// TIA Portal V17 export
// export: Created 2023-02-26T22:59:49.9931463Z, ExportSetting WithDefaults, DisplayName Totally Integrated Automation Portal, DisplayVersion V17, DisplayName TIA Portal Openness, DisplayVersion V17, DisplayName TIA Portal Version Control Interface, DisplayVersion V17, DisplayName TIA Portal Test Suite Advanced, DisplayVersion V17, DisplayName STEP 7 Professional, DisplayVersion V17, DisplayName SIMATIC Energy Suite, DisplayVersion V17, DisplayName STEP 7 Safety, DisplayVersion V17, DisplayName WinCC Professional, DisplayVersion V17
FUNCTION "LOG_ConveyorTime" : Void   // FC20, LAD
{ S7_Optimized_Access := 'TRUE' }
VERSION : 0.1
// stored: AutoNumber true, IsIECCheckEnabled false, SetENOAutomatically false, UDAEnableTagReadback false
   VAR_TEMP
      t_RisingTime : Bool;
   END_VAR
BEGIN

REGION Network 1: Trigger
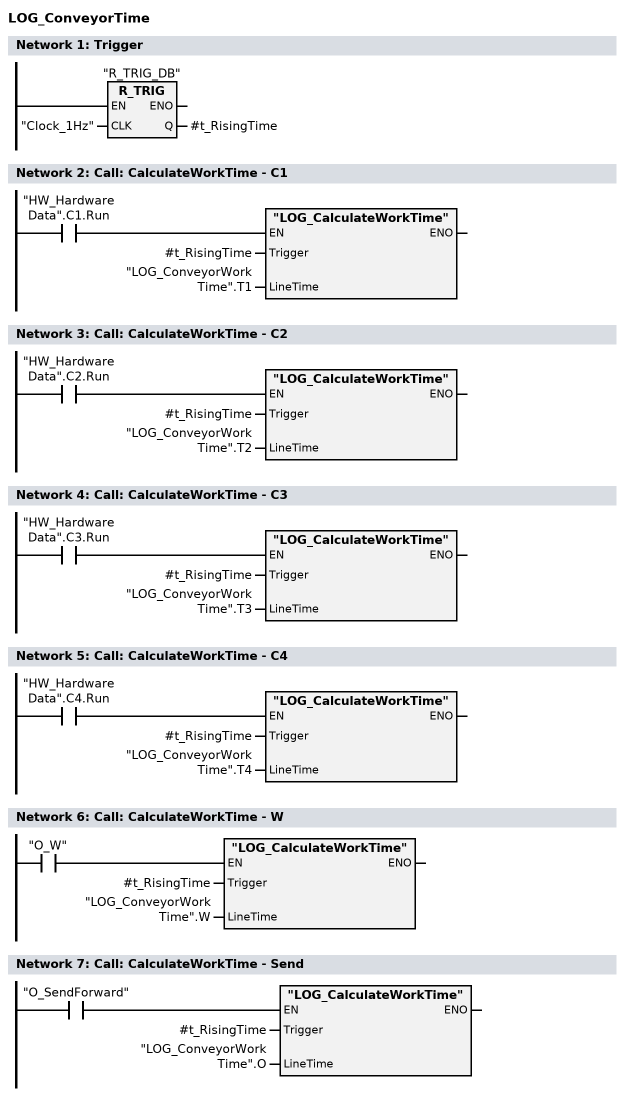
   RUNG wire#powerrail
      "R_TRIG_DB".R_TRIG(CLK := "Clock_1Hz", Q => #t_RisingTime)
   END_RUNG
   // the same network as SCL:
   "R_TRIG_DB"(CLK := "Clock_1Hz", Q => #t_RisingTime);   // R_TRIG
END_REGION

REGION Network 2: Call: CalculateWorkTime - C1
   RUNG wire#powerrail
      Contact( "HW_HardwareData".C1.Run )
      "LOG_CalculateWorkTime"(Trigger := #t_RisingTime, LineTime := "LOG_ConveyorWorkTime".T1)
   END_RUNG
   // the same network as SCL:
   IF "HW_HardwareData".C1.Run THEN
       "LOG_CalculateWorkTime"(Trigger := #t_RisingTime, LineTime := "LOG_ConveyorWorkTime".T1);
   END_IF;
END_REGION

REGION Network 3: Call: CalculateWorkTime - C2
   RUNG wire#powerrail
      Contact( "HW_HardwareData".C2.Run )
      "LOG_CalculateWorkTime"(Trigger := #t_RisingTime, LineTime := "LOG_ConveyorWorkTime".T2)
   END_RUNG
   // the same network as SCL:
   IF "HW_HardwareData".C2.Run THEN
       "LOG_CalculateWorkTime"(Trigger := #t_RisingTime, LineTime := "LOG_ConveyorWorkTime".T2);
   END_IF;
END_REGION

REGION Network 4: Call: CalculateWorkTime - C3
   RUNG wire#powerrail
      Contact( "HW_HardwareData".C3.Run )
      "LOG_CalculateWorkTime"(Trigger := #t_RisingTime, LineTime := "LOG_ConveyorWorkTime".T3)
   END_RUNG
   // the same network as SCL:
   IF "HW_HardwareData".C3.Run THEN
       "LOG_CalculateWorkTime"(Trigger := #t_RisingTime, LineTime := "LOG_ConveyorWorkTime".T3);
   END_IF;
END_REGION

REGION Network 5: Call: CalculateWorkTime - C4
   RUNG wire#powerrail
      Contact( "HW_HardwareData".C4.Run )
      "LOG_CalculateWorkTime"(Trigger := #t_RisingTime, LineTime := "LOG_ConveyorWorkTime".T4)
   END_RUNG
   // the same network as SCL:
   IF "HW_HardwareData".C4.Run THEN
       "LOG_CalculateWorkTime"(Trigger := #t_RisingTime, LineTime := "LOG_ConveyorWorkTime".T4);
   END_IF;
END_REGION

REGION Network 6: Call: CalculateWorkTime - W
   RUNG wire#powerrail
      Contact( "O_W" )
      "LOG_CalculateWorkTime"(Trigger := #t_RisingTime, LineTime := "LOG_ConveyorWorkTime".W)
   END_RUNG
   // the same network as SCL:
   IF "O_W" THEN
       "LOG_CalculateWorkTime"(Trigger := #t_RisingTime, LineTime := "LOG_ConveyorWorkTime".W);
   END_IF;
END_REGION

REGION Network 7: Call: CalculateWorkTime - Send
   RUNG wire#powerrail
      Contact( "O_SendForward" )
      "LOG_CalculateWorkTime"(Trigger := #t_RisingTime, LineTime := "LOG_ConveyorWorkTime".O)
   END_RUNG
   // the same network as SCL:
   IF "O_SendForward" THEN
       "LOG_CalculateWorkTime"(Trigger := #t_RisingTime, LineTime := "LOG_ConveyorWorkTime".O);
   END_IF;
END_REGION
END_FUNCTION
